FUNCTION_BLOCK FB_Teltonika

VAR_IN_OUT CONSTANT
	st_params	: st_Router_Params;
END_VAR

VAR_IN_OUT
	st_service : ST_router_service;
END_VAR

VAR
	realconverter : dwtoreal;
	w_SendSMS: WORD;
	set : st_router_set;
	ui_counter	:	uint;
END_VAR
VAR_OUTPUT
	Get	:	st_router_get;
END_VAR
VAR
	MBRead			: 	FB_MBReadRegs;
	MBWrite			:	FB_MBWriteRegs;
	MBSingleWrite	:	FB_MBWriteSingleReg;
	
	arw_DataBuffer		: 	ARRAY[0..62] OF word;
	st_WriteSMSData		:	STRING(20);

	ar_SMSData			:	ARRAY[0..89] OF WORD;
	ar_ReadSMSData		:	ARRAY[0..89] OF WORD;
	
	tempbuffer			:	ARRAY[0..10] OF WORD;

	
	ton_GetDataTimer				:	TON := (PT := TIME#1000MS);
	ton_StartSMSServiceDelay		:	TON := (PT := T#60S);

	
	ftrig_TransmissionDone	:	F_trig;
	
	ui_MBRetryCount			:	UINT;
	ui_SMSRetryCounter	:	UINT;
		
	ui_ForCounter	:	UINT;
	ui_MessageCounter	:	UINT;
	b_busy: BOOL;
	b_CommError: BOOL;
	udi_errid: UDINT;
	udi_cbread: UDINT;
	
	
	TempDTString	:	String;
END_VAR


VAR_IN_OUT
	s_Message	:	ARRAY[*] OF STRING;
END_VAR

VAR_INPUT
	s_SerialNumber		: STRING;
END_VAR

VAR CONSTANT
	e_ID 				: eObject_ID := eObject_ID.Router;
END_VAR

ton_GetDataTimer(IN:=NOT ton_GetDataTimer.Q);
ton_StartSMSServiceDelay();

ReadDataSFC();

get.Events.b_MBCommWarning := ui_MBRetryCount > 20;


//temporary setup via stparams until hmi setup is implemented.
set := st_params.ManualSettings;

ACTION aCheckAlarmMessages:
IF ton_StartSMSServiceDelay.Q THEN
	IF get.e_SMSStatus = eSMSStatus.Idle OR get.e_SMSStatus = eSMSStatus.error THEN
		//skip through message array until non_empty value or the end of the list is found 
		WHILE (s_Message[ui_MessageCounter] = '') AND (ui_MessageCounter < UPPER_BOUND(s_message, 1)) DO
			ui_MessageCounter := ui_MessageCounter + 1;
		END_WHILE
		
		IF (s_Message[ui_MessageCounter] <> '') THEN
			CreateMessage(s_Message[ui_MessageCounter]);	//check for valid message
			get.e_SMSStatus := eSMSStatus.NewMessage;
			s_Message[ui_MessageCounter] := '';
		END_IF
		
		IF ui_MessageCounter >= UPPER_BOUND(s_message, 1) THEN
			ui_MessageCounter := DINT_TO_UINT(LOWER_BOUND(s_message, 1)); 
		END_IF
	END_IF
END_IF
END_ACTION

ACTION aNetworkinfo:
MBRead(
	sIPAddr := st_params.IP_TELTONIKA,
	nTCPPort := st_params.MBPort_TELTONIKA,
	nUnitID := 1,
	nMBAddr := 103,
	nQuantity := 32,//*2,
	cbLength := SIZEOF(arw_DataBuffer),
	pDestAddr := ADR(arw_DataBuffer),
	bExecute := ton_GetDataTimer.Q,
	bBusy => b_busy,
	bError => b_CommError,
	nErrId => udi_errid,
	cbRead => udi_cbread,
	tTimeout := st_params.T_MBTimeout
);

ftrig_TransmissionDone(clk := b_busy);

IF ftrig_TransmissionDone.q THEN
	IF NOT b_CommError THEN
		FOR ui_ForCounter := 0 TO 31 DO
			arw_DataBuffer[ui_ForCounter] := be16_TO_HOST(arw_DataBuffer[ui_ForCounter]);
		END_FOR
		
		MEMCPY(ADR(Get.Mobile.NetworkInfo),  ADR(arw_DataBuffer[0]), 32);
		MEMCPY(ADR(Get.Mobile.NetworkType),  ADR(arw_DataBuffer[16]), 32);
		ui_MBRetryCount := 0;
		sfctip := TRUE;
	ELSE
		ui_MBRetryCount := ui_MBRetryCount + 1;
		sfctip := TRUE;
	END_IF
END_IF
END_ACTION

ACTION aReadActiveSim:

MBRead(
	sIPAddr := st_params.IP_TELTONIKA,
	nTCPPort := st_params.MBPort_TELTONIKA,
	nUnitID := 1,
	nMBAddr := 205,
	nQuantity := 1,//*2,
	cbLength := SIZEOF(arw_DataBuffer),
	pDestAddr := ADR(arw_DataBuffer),
	bExecute := ton_GetDataTimer.Q,
	bBusy => b_busy,
	bError => b_CommError,
	nErrId => udi_errid,
	cbRead => udi_cbread,
	tTimeout := st_params.T_MBTimeout
);

ftrig_TransmissionDone(clk := b_busy);

IF ftrig_TransmissionDone.q THEN
	IF NOT b_CommError THEN
	
		//Get.Mobile.ui_ActiveSim := arw_DataBuffer[0];
	
		ui_MBRetryCount := 0;
		sfctip := TRUE;
	ELSE
		ui_MBRetryCount := ui_MBRetryCount + 1;
		sfctip := TRUE;
	END_IF
END_IF
END_ACTION

ACTION aReadDataUsageSim1:

MBRead(
	sIPAddr := st_params.IP_TELTONIKA,
	nTCPPort := st_params.MBPort_TELTONIKA,
	nUnitID := 1,
	nMBAddr := 193,
	nQuantity := 4,//*2,
	cbLength := SIZEOF(arw_DataBuffer),
	pDestAddr := ADR(arw_DataBuffer),
	bExecute := ton_GetDataTimer.Q,
	bBusy => b_busy,
	bError => b_CommError,
	nErrId => udi_errid,
	cbRead => udi_cbread,
	tTimeout := st_params.T_MBTimeout
);

ftrig_TransmissionDone(clk := b_busy);

IF ftrig_TransmissionDone.q THEN
	IF NOT b_CommError THEN
	
		MEMCPY(ADR(Get.Mobile.ui_Sim1DataReceivedMonth)+2, ADR(arw_DataBuffer[0]), 2);
		MEMCPY(ADR(Get.Mobile.ui_Sim1DataReceivedMonth), ADR(arw_DataBuffer[1]), 2);
		
		MEMCPY(ADR(Get.Mobile.ui_Sim1DataSendMonth)+2, ADR(arw_DataBuffer[2]), 2);
		MEMCPY(ADR(Get.Mobile.ui_Sim1DataSendMonth), ADR(arw_DataBuffer[3]), 2);	
	
		ui_MBRetryCount := 0;
		sfctip := TRUE;
	ELSE
		ui_MBRetryCount := ui_MBRetryCount + 1;
		sfctip := TRUE;
	END_IF
END_IF
END_ACTION

ACTION aReadDataUsageSim2:

MBRead(
	sIPAddr := st_params.IP_TELTONIKA,
	nTCPPort := st_params.MBPort_TELTONIKA,
	nUnitID := 1,
	nMBAddr := 308,
	nQuantity := 4,//*2,
	cbLength := SIZEOF(arw_DataBuffer),
	pDestAddr := ADR(arw_DataBuffer),
	bExecute := ton_GetDataTimer.Q,
	bBusy => b_busy,
	bError => b_CommError,
	nErrId => udi_errid,
	cbRead => udi_cbread,
	tTimeout := st_params.T_MBTimeout
);

ftrig_TransmissionDone(clk := b_busy);

IF ftrig_TransmissionDone.q THEN
	IF NOT b_CommError THEN
	
		MEMCPY(ADR(Get.Mobile.ui_Sim2DataReceivedMonth)+2, ADR(arw_DataBuffer[0]), 2);
		MEMCPY(ADR(Get.Mobile.ui_Sim2DataReceivedMonth), ADR(arw_DataBuffer[1]), 2);
		
		MEMCPY(ADR(Get.Mobile.ui_Sim2DataSendMonth)+2, ADR(arw_DataBuffer[2]), 2);
		MEMCPY(ADR(Get.Mobile.ui_Sim2DataSendMonth), ADR(arw_DataBuffer[3]), 2);	
	
		ui_MBRetryCount := 0;
		sfctip := TRUE;
	ELSE
		ui_MBRetryCount := ui_MBRetryCount + 1;
		sfctip := TRUE;
	END_IF
END_IF
END_ACTION

ACTION AReadGeneral:

MBRead(
	sIPAddr := st_params.IP_TELTONIKA,
	nTCPPort := st_params.MBPort_TELTONIKA,
	nUnitID := 1,
	nMBAddr := 1,
	nQuantity := 6,//*2,
	cbLength := SIZEOF(arw_DataBuffer),
	pDestAddr := ADR(arw_DataBuffer),
	bExecute := ton_GetDataTimer.Q,
	bBusy => b_busy,
	bError => b_CommError,
	nErrId => udi_errid,
	cbRead => udi_cbread,
	tTimeout := st_params.T_MBTimeout
);

ftrig_TransmissionDone(clk := b_busy);

IF ftrig_TransmissionDone.q THEN
	IF NOT b_CommError THEN
		
		get.Device.SystemUptime :=	SHL(	WORD_TO_UDINT(	arw_DataBuffer[0]),16)	+	arw_DataBuffer[1];
		MEMCPY(ADR(Get.Mobile.RSSI)+2,  ADR(arw_DataBuffer[2]), 2);
		MEMCPY(ADR(Get.Mobile.RSSI),  ADR(arw_DataBuffer[3]), 2);

		//MEMCPY(ADR(Get.Mobile.NetworkOperator),  ADR(arw_DataBuffer[22]), 32);
		
		get.Device.Temperature	:= 	UDINT_TO_REAL ( SHL(	WORD_TO_UDINT(	arw_DataBuffer[4]),16)	+	arw_DataBuffer[5] )/10;

		ui_MBRetryCount := 0;
		sfctip := TRUE;
	ELSE
		ui_MBRetryCount := ui_MBRetryCount + 1;
		sfctip := TRUE;
	END_IF
END_IF
END_ACTION

ACTION aReadGPSData:


MBRead(
	sIPAddr := st_params.IP_TELTONIKA,
	nTCPPort := st_params.MBPort_TELTONIKA,
	nUnitID := 1,
	nMBAddr := 143,
	nQuantity := 42,//*2,
	cbLength := SIZEOF(arw_DataBuffer),
	pDestAddr := ADR(arw_DataBuffer),
	bExecute := ton_GetDataTimer.Q,
	bBusy => b_busy,
	bError => b_CommError,
	nErrId => udi_errid,
	cbRead => udi_cbread,
	tTimeout := st_params.T_MBTimeout
);

ftrig_TransmissionDone(clk := b_busy);

IF ftrig_TransmissionDone.q THEN
	IF NOT b_CommError THEN
		
		realconverter.Registers[2] := arw_DataBuffer[0];
		realconverter.Registers[1] := arw_DataBuffer[1];
		Get.GPS.Latitude  := realconverter.realvalue;
 
		realconverter.Registers[2] := arw_DataBuffer[2];
		realconverter.Registers[1] := arw_DataBuffer[3];
		Get.GPS.Longitude  := realconverter.realvalue;
		
		FOR ui_ForCounter := 4 TO 35 DO
			arw_DataBuffer[ui_ForCounter] := be16_TO_HOST(arw_DataBuffer[ui_ForCounter]);
		END_FOR
				
		MEMCPY(ADR(Get.GPS.FixTime),  ADR(arw_DataBuffer[4]), 32);			//GPS fixtime (text, unix timetamp * 1000)
						
		MEMCPY(ADR(TempDTString), ADR(arw_DataBuffer[20]), 32);			//GPS DateTime (text, YYYY-MM-DD HH:MM:SS)
		FindAndReplaceChar(ADR(TempDTString), ' ', '-', ADR(TempDTString), SIZEOF(TempDTString));	//replace space between date and time with dash
		TempDTString := concat(TempDTString, '.000');	//add milliseconds to string
		get.GPS.DateTime := SystemTime_TO_DT(String_TO_Systemtime(TempDTString));
		
		realconverter.Registers[2] := arw_DataBuffer[36];					//GPS speed
		realconverter.Registers[1] := arw_DataBuffer[37];
		Get.GPS.Speed  := realconverter.realvalue;
		
	
		MEMCPY(ADR(Get.GPS.SatCount)+2, ADR(arw_DataBuffer[38]), 2);			//GPS sattelite count
		MEMCPY(ADR(Get.GPS.SatCount), ADR(arw_DataBuffer[39]), 2);			//GPS sattelite count
		
		realconverter.Registers[2] := arw_DataBuffer[40];
		realconverter.Registers[1] := arw_DataBuffer[41];
		Get.GPS.Accuracy  := realconverter.realvalue;						//GPS accuracy
		
			
		ui_MBRetryCount := 0;
		sfctip := TRUE;
	ELSE
		ui_MBRetryCount := ui_MBRetryCount + 1;
		sfctip := TRUE;
	END_IF
END_IF
END_ACTION

ACTION aReadSerial:
MBRead(
	sIPAddr := st_params.IP_TELTONIKA,
	nTCPPort := st_params.MBPort_TELTONIKA,
	nUnitID := 1,
	nMBAddr := 39,
	nQuantity := 16,//*2,
	cbLength := SIZEOF(arw_DataBuffer),
	pDestAddr := ADR(arw_DataBuffer),
	bExecute := ton_GetDataTimer.Q,
	bBusy => b_busy,
	bError => b_CommError,
	nErrId => udi_errid,
	cbRead => udi_cbread,
	tTimeout := st_params.T_MBTimeout
);

ftrig_TransmissionDone(clk := b_busy);

IF ftrig_TransmissionDone.q THEN
	IF NOT b_CommError THEN
		FOR ui_ForCounter := 0 TO 16 DO
			arw_DataBuffer[ui_ForCounter] := be16_TO_HOST(arw_DataBuffer[ui_ForCounter]);
		END_FOR
		
		//MEMCPY(ADR(Get.Mobile.NetworkOperator),  ADR(arw_DataBuffer[0]), 32);
		MEMCPY(ADR(Get.Device.RouterSerial),  ADR(arw_DataBuffer[0]), 32);
		
		ui_MBRetryCount := 0;
		sfctip := TRUE;
	ELSE
		ui_MBRetryCount := ui_MBRetryCount + 1;
		sfctip := TRUE;
	END_IF
END_IF
END_ACTION

ACTION aSendSMS:

IF get.e_SMSStatus = eSMSStatus.SendingMessage THEN
	MBSingleWrite(
		sIPAddr := st_params.IP_TELTONIKA,
		nTCPPort := st_params.MBPort_TELTONIKA,
		nUnitID := 1,
		nMBAddr := 396,
		nValue	:=	1,
		bExecute := ton_GetDataTimer.Q,
		bBusy => b_busy,
		bError => b_CommError,
		nErrId => udi_errid,
		tTimeout := st_params.T_MBTimeout
	);
	
	ftrig_TransmissionDone(clk := b_busy);
	
	IF ftrig_TransmissionDone.q THEN
		IF NOT b_CommError THEN
			get.e_SMSStatus := eSMSSTatus.idle;		
			ui_SMSRetryCounter := 0;
			ui_MBRetryCount := 0;
			sfctip := TRUE;
		ELSE
			ui_MBRetryCount := ui_MBRetryCount + 1;
			ui_SMSRetryCounter := ui_SMSRetryCounter + 1;
			IF ui_SMSRetryCounter > 0 THEN
				get.Events.b_SMSNotSendError := TRUE;
				get.e_SMSStatus := eSMSStatus.error;
				sfctip := TRUE;
			END_IF
		END_IF
	END_IF
ELSE
	SFCtip := NOT SFCTip;
END_IF
END_ACTION

ACTION aWriteSimSettings:

arw_DataBuffer[0] := TO_UINT(set.SimSelectionMode);
arw_DataBuffer[1] := TO_UINT(set.Sim1Pin);
arw_DataBuffer[2] := TO_UINT(set.Sim2Pin);

//FOR ui_counter := 1 TO 3 DO
//	arw_DataBuffer[ui_counter] := host_to_be16(arw_DataBuffer[ui_counter]);
//END_FOR

MBWrite(
	sIPAddr := st_params.IP_TELTONIKA,
	nTCPPort := st_params.MBPort_TELTONIKA,
	nUnitID := 1,
	nMBAddr := 1049,
	nQuantity := 3,
	cbLength := SIZEOF(arw_DataBuffer),
	pSrcAddr	:=	ADR(arw_DataBuffer),
	bExecute := ton_GetDataTimer.Q,
	bBusy => b_busy,
	bError => b_CommError,
	nErrId => udi_errid,
	tTimeout := st_params.T_MBTimeout
);

ftrig_TransmissionDone(clk := b_busy);

IF ftrig_TransmissionDone.q THEN
		sfctip := TRUE;
END_IF
END_ACTION

ACTION aWriteSMSData:

MBWrite(
	sIPAddr := st_params.IP_TELTONIKA,
	nTCPPort := st_params.MBPort_TELTONIKA,
	nUnitID := 1,
	nMBAddr := 397,
	nQuantity := 90,
	cbLength := SIZEOF(ar_SMSData),
	pSrcAddr	:=	ADR(ar_SMSData),
	bExecute := ton_GetDataTimer.Q,
	bBusy => b_busy,
	bError => b_CommError,
	nErrId => udi_errid,
	tTimeout := st_params.T_MBTimeout
);

ftrig_TransmissionDone(clk := b_busy);

IF ftrig_TransmissionDone.q THEN
	IF NOT b_CommError THEN
		get.e_SMSStatus := eSMSStatus.SendingMessage;
		ui_SMSRetryCounter := 0;
		ui_MBRetryCount := 0;
		sfctip := TRUE;
	ELSE
		ui_SMSRetryCounter := ui_SMSRetryCounter +1;
		ui_MBRetryCount := ui_MBRetryCount + 1;
		IF ui_SMSRetryCounter > 3 THEN
			get.Events.b_SMSNotSendError := TRUE;
			get.e_SMSStatus := eSMSStatus.error;
			sfctip := TRUE;
		END_IF
	END_IF
END_IF
END_ACTION

ACTION Bypass_active:
get.e_SMSStatus := eSMSStatus.Idle;
get.Events.b_SMSNotSendError := FALSE;
END_ACTION

METHOD CreateMessage : BOOL
VAR_INPUT
//	TelNumber	:	ULINT;
	s_Message		:	STRING(80);
END_VAR

VAR
	s_InternalMessage 	: 	STRING(160);
	s_LAT				:	STRING(8);
	s_LONG				:	STRING(9);
	ui_counter			:	UINT;
END_VAR
IF NOT get.Events.b_NoSMSNumberAvailable THEN
	memcpy(ADR(ar_SMSData[0]), ADR(get.Mobile.s_EmergencySMSNumber), 20);
	
	s_LAT := REAL_TO_STRING(get.GPS.Latitude);
	s_LONG := REAL_TO_STRING(get.GPS.Longitude);
	
	s_InternalMessage := 'ePU10 LFP Battery System';
	s_InternalMessage := concat(s_InternalMessage, '$n');
	s_InternalMessage := concat(s_InternalMessage, 'ID: ');
	s_InternalMessage := concat(s_InternalMessage, get.mobile.s_EmergencySMSDevName);
	s_InternalMessage := concat(s_InternalMessage, '$n');
	s_InternalMessage := concat(s_InternalMessage, 'LAT: ');
	s_InternalMessage := concat(s_InternalMessage, s_LAT);
	s_InternalMessage := concat(s_InternalMessage, '$n');
	s_InternalMessage := concat(s_InternalMessage, 'LON: ');
	s_InternalMessage := concat(s_InternalMessage, s_LONG);
	s_InternalMessage := concat(s_InternalMessage, '$n');
	s_InternalMessage := concat(s_InternalMessage,s_Message);
	
	memcpy(ADR(ar_SMSData[10]), ADR(s_InternalMessage[0]), 160);
	
	FOR ui_counter := 0 TO 89 DO
		ar_SMSData[ui_counter] := host_to_be16(ar_SMSData[ui_counter]);
	END_FOR

	CreateMessage := TRUE;
ELSE
	get.Events.b_SMSNotSendError := TRUE;
	CreateMessage := TRUE;
END_IF
END_METHOD

METHOD EMStop : BOOL
VAR_INPUT
END_VAR

//nothing to do here
EMSTOP := TRUE;
END_METHOD

METHOD FB_init : BOOL
VAR_INPUT
	bInitRetains : BOOL; // if TRUE, the retain variables are initialized (warm start / cold start)
	bInCopyCode : BOOL;  // if TRUE, the instance afterwards gets moved into the copy code (online change)
END_VAR
ton_StartSMSServiceDelay(IN := TRUE);
END_METHOD

METHOD GetDiagnostics : BOOL
VAR_IN_OUT
	AddError		: ARRAY [*] OF FB_AddErrorST;
	a_ActiveEvents	: ARRAY [*] OF ST_ErrorStruct;
	w_Index			: WORD;
END_VAR
(*No emergency number configured*)	AddError[w_Index](
			b_ErrorTrig				:= get.Events.b_NoSMSNumberAvailable,
			b_SMSEnableVDL			:= FALSE,
			out_ST_Error			:= a_ActiveEvents[w_Index],
			w_ErrorID				:= 1,
			e_ObjectID				:= e_id,						//only first call set object ID.
			s_Message				:= 'no sms number available',
			e_sev					:= eSeverity.info,
			b_AutoClear				:= TRUE,
			e_ErrAckAccess			:= eErrAckAccess.General
			);
		w_Index := w_Index +1;
		
(*SMS not send warning*)	AddError[w_Index](
			b_ErrorTrig				:= get.Events.b_SMSNotSendError,
			b_SMSEnableVDL			:= FALSE,
			out_ST_Error			:= a_ActiveEvents[w_Index],
			w_ErrorID				:= 2,					
			s_Message				:= 'SMS not send',
			e_sev					:= eSeverity.info,
			b_AutoClear				:= TRUE,
			t_triggerTime			:= T#10S,
			e_ErrAckAccess			:= eErrAckAccess.General
			);
		w_Index := w_Index +1;
		
(*Modbus comm warning*)	AddError[w_Index](
			b_ErrorTrig				:= get.Events.b_MBCommWarning,
			b_SMSEnableVDL			:= FALSE,
			out_ST_Error			:= a_ActiveEvents[w_Index],
			w_ErrorID				:= 3,					
			s_Message				:= 'modbus comm. warning',
			e_sev					:= eSeverity.warning,
			b_AutoClear				:= TRUE,
			e_ErrAckAccess			:= eErrAckAccess.General
			);
		w_Index := w_Index +1;
		
(*GPS location missing*)	AddError[w_Index](
			b_ErrorTrig				:= get.Events.b_noGPSFixWarning,
			b_SMSEnableVDL			:= FALSE,
			out_ST_Error			:= a_ActiveEvents[w_Index],
			w_ErrorID				:= 5,					
			s_Message				:= 'no gps location available',
			e_sev					:= eSeverity.info,
			b_AutoClear				:= TRUE,
			e_ErrAckAccess			:= eErrAckAccess.General
			);
		w_Index := w_Index +1;
		
(*network missing*)	AddError[w_Index](
			b_ErrorTrig				:= get.Events.b_NoNetworkWarning,
			b_SMSEnableVDL			:= FALSE,
			out_ST_Error			:= a_ActiveEvents[w_Index],
			w_ErrorID				:= 6,					
			s_Message				:= 'no network available',
			e_sev					:= eSeverity.info,
			b_AutoClear				:= TRUE,
			e_ErrAckAccess			:= eErrAckAccess.General
			);
		w_Index := w_Index +1;
		
(*simcard missing*)	AddError[w_Index](
			b_ErrorTrig				:= get.Events.b_NoSimWarning,
			b_SMSEnableVDL			:= FALSE,
			out_ST_Error			:= a_ActiveEvents[w_Index],
			w_ErrorID				:= 7,					
			s_Message				:= 'no simcard available',
			e_sev					:= eSeverity.info,
			b_AutoClear				:= TRUE,
			e_ErrAckAccess			:= eErrAckAccess.General
			);
		w_Index := w_Index +1;
END_METHOD

ACTION ReadCustomRegisters:

MBRead(
	sIPAddr := st_params.IP_TELTONIKA,
	nTCPPort := st_params.MBPort_TELTONIKA,
	nUnitID := 1,
	nMBAddr := 1024,
	nQuantity := 7,//*2,
	cbLength := SIZEOF(arw_DataBuffer),
	pDestAddr := ADR(arw_DataBuffer),
	bExecute := ton_GetDataTimer.Q,
	bBusy => b_busy,
	bError => b_CommError,
	nErrId => udi_errid,
	cbRead => udi_cbread,
	tTimeout := st_params.T_MBTimeout
);

ftrig_TransmissionDone(clk := b_busy);

IF ftrig_TransmissionDone.q THEN
	IF NOT b_CommError THEN
		get.Mobile.ui_ActiveSim 		:= 	arw_DataBuffer[0];
		get.Mobile.SimStatus 			:= 	arw_DataBuffer[1];
		get.Mobile.ModemState 			:= 	arw_DataBuffer[2];
		get.Mobile.NetworkState 		:=  arw_DataBuffer[3];
		get.Wifi.WifiClienModeStatus 	:= 	arw_DataBuffer[4]; 
		get.Wifi.WifiAPModeStatus 		:= 	arw_DataBuffer[5]; 		//not yet implemented
		get.Wifi.WifiApNumberOfClients 	:= 	arw_DataBuffer[6]; 
		
			
		ui_MBRetryCount := 0;
		sfctip := TRUE;
	ELSE
		ui_MBRetryCount := ui_MBRetryCount + 1;
		sfctip := TRUE;
	END_IF
END_IF
END_ACTION

ACTION ReadDataSFC:
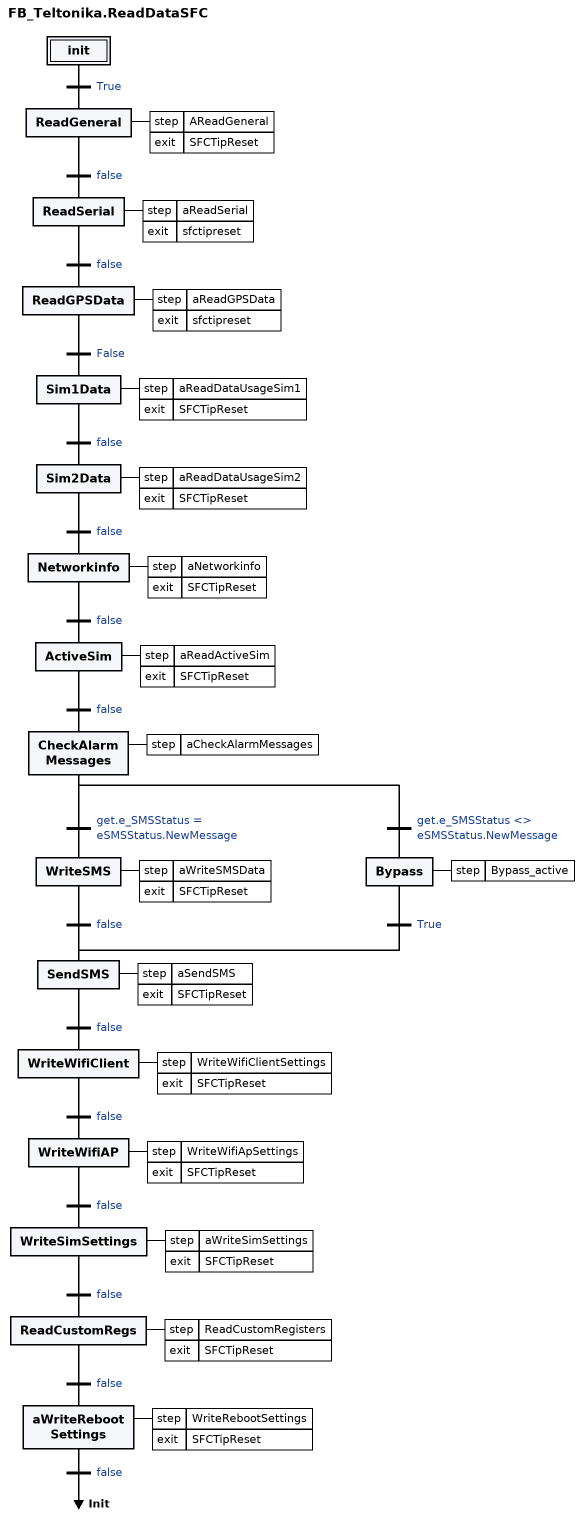
INITIAL_STEP init:
END_STEP
TRANSITION FROM init TO ReadGeneral
    := True;
END_TRANSITION
STEP ReadGeneral:
    AReadGeneral(N);  // step action
    SFCTipReset(P0);  // exit action
END_STEP
TRANSITION FROM ReadGeneral TO ReadSerial
    := false;
END_TRANSITION
STEP ReadSerial:
    aReadSerial(N);  // step action
    sfctipreset(P0);  // exit action
END_STEP
TRANSITION FROM ReadSerial TO ReadGPSData
    := false;
END_TRANSITION
STEP ReadGPSData:
    aReadGPSData(N);  // step action
    sfctipreset(P0);  // exit action
END_STEP
TRANSITION FROM ReadGPSData TO Sim1Data
    := False;
END_TRANSITION
STEP Sim1Data:
    aReadDataUsageSim1(N);  // step action
    SFCTipReset(P0);  // exit action
END_STEP
TRANSITION FROM Sim1Data TO Sim2Data
    := false;
END_TRANSITION
STEP Sim2Data:
    aReadDataUsageSim2(N);  // step action
    SFCTipReset(P0);  // exit action
END_STEP
TRANSITION FROM Sim2Data TO Networkinfo
    := false;
END_TRANSITION
STEP Networkinfo:
    aNetworkinfo(N);  // step action
    SFCTipReset(P0);  // exit action
END_STEP
TRANSITION FROM Networkinfo TO ActiveSim
    := false;
END_TRANSITION
STEP ActiveSim:
    aReadActiveSim(N);  // step action
    SFCTipReset(P0);  // exit action
END_STEP
TRANSITION FROM ActiveSim TO CheckAlarmMessages
    := false;
END_TRANSITION
STEP CheckAlarmMessages:
    aCheckAlarmMessages(N);  // step action
END_STEP
TRANSITION FROM CheckAlarmMessages TO WriteSMS
    := get.e_SMSStatus = eSMSStatus.NewMessage;
END_TRANSITION
STEP WriteSMS:
    aWriteSMSData(N);  // step action
    SFCTipReset(P0);  // exit action
END_STEP
TRANSITION FROM WriteSMS TO SendSMS
    := false;
END_TRANSITION
TRANSITION FROM CheckAlarmMessages TO Bypass
    := get.e_SMSStatus <> eSMSStatus.NewMessage;
END_TRANSITION
STEP Bypass:
    Bypass_active(N);  // step action
END_STEP
TRANSITION FROM Bypass TO SendSMS
    := True;
END_TRANSITION
STEP SendSMS:
    aSendSMS(N);  // step action
    SFCTipReset(P0);  // exit action
END_STEP
TRANSITION FROM SendSMS TO WriteWifiClient
    := false;
END_TRANSITION
STEP WriteWifiClient:
    WriteWifiClientSettings(N);  // step action
    SFCTipReset(P0);  // exit action
END_STEP
TRANSITION FROM WriteWifiClient TO WriteWifiAP
    := false;
END_TRANSITION
STEP WriteWifiAP:
    WriteWifiApSettings(N);  // step action
    SFCTipReset(P0);  // exit action
END_STEP
TRANSITION FROM WriteWifiAP TO WriteSimSettings
    := false;
END_TRANSITION
STEP WriteSimSettings:
    aWriteSimSettings(N);  // step action
    SFCTipReset(P0);  // exit action
END_STEP
TRANSITION FROM WriteSimSettings TO ReadCustomRegs
    := false;
END_TRANSITION
STEP ReadCustomRegs:
    ReadCustomRegisters(N);  // step action
    SFCTipReset(P0);  // exit action
END_STEP
TRANSITION FROM ReadCustomRegs TO aWriteRebootSettings
    := false;
END_TRANSITION
STEP aWriteRebootSettings:
    WriteRebootSettings(N);  // step action
    SFCTipReset(P0);  // exit action
END_STEP
TRANSITION FROM aWriteRebootSettings TO Init
    := false;
END_TRANSITION
// branch label Branch0_ReadDataSFC
END_ACTION

METHOD Reset : BOOL
VAR_INPUT
END_VAR
get.Events.b_SMSNotSendError := FALSE;
get.e_SMSStatus := eSMSStatus.Idle;

Reset := TRUE;
END_METHOD

METHOD SetDevName : BOOL
VAR_INPUT
	s_DevName	:	String(12);
END_VAR
IF s_DevName = '' THEN
	get.Mobile.s_EmergencySMSDevName := ''; //<-- stParams.serial number
ELSE
	get.Mobile.s_EmergencySMSDevName :=	s_DevName;
END_IF

SetDevName := get.Mobile.s_EmergencySMSDevName <> '';
END_METHOD

METHOD SetSMSNumber : BOOL
VAR_INPUT
	s_SMSNumber	:	STRING(20);
END_VAR
VAR 
	for_counter	:	UINT :=0;
	InternalString	:	STRING(20);
	intermediateValue	:	UINT;
	
	temp	:	string(10);
END_VAR

SetSMSNumber := TRUE;

//check minimum length
IF INT_TO_UINT(len(s_SMSNumber)) < st_params.MinimumPhoneNumberLength AND s_SMSNumber <> '' THEN
	SetSMSNumber := FALSE;
ELSE
	InternalString := s_SMSNumber;
	
	//replace leading + with 00
	IF left(InternalString,1) = '+' THEN
		InternalString := Replace(InternalString, '00', 1, 1);
	END_IF
	
	//check for non_numeric characters
	FOR for_counter := 1 TO INT_TO_UINT(len(InternalString)) DO
		intermediateValue := f_toASC(mid(InternalString, 1, UINT_TO_INT(for_counter)));
		IF (intermediateValue < 48 OR intermediateValue > 57) THEN
			SetSMSNumber := FALSE;
		END_IF
	END_FOR
END_IF

//only if all checks succeed, the number is written to the struct.
IF SetSMSNumber THEN
	get.Mobile.s_EmergencySMSNumber := InternalString;
ELSE
	get.Mobile.s_EmergencySMSNumber := '';
END_IF

get.Events.b_NoSMSNumberAvailable := NOT SetSMSNumber;
END_METHOD

ACTION SFCTipReset:
SFCTip := FALSE;
END_ACTION

ACTION WriteRebootSettings:

arw_DataBuffer[0] := TO_UINT(set.AutoRebootEnable);
arw_DataBuffer[1] := TO_UINT(set.ManualReboot);

MBWrite(
	sIPAddr := st_params.IP_TELTONIKA,
	nTCPPort := st_params.MBPort_TELTONIKA,
	nUnitID := 1,
	nMBAddr := 1139,
	nQuantity := 2,
	cbLength := SIZEOF(arw_DataBuffer),
	pSrcAddr	:=	ADR(arw_DataBuffer),
	bExecute := ton_GetDataTimer.Q,
	bBusy => b_busy,
	bError => b_CommError,
	nErrId => udi_errid,
	tTimeout := st_params.T_MBTimeout
);

ftrig_TransmissionDone(clk := b_busy);

IF ftrig_TransmissionDone.q THEN
	sfctip := TRUE;
	set.ManualReboot := false;
END_IF
END_ACTION

ACTION WriteWifiAPSettings:

arw_DataBuffer[0] := TO_UINT(set.EnableWifiAP);
memcpy(ADR(arw_DataBuffer[1]), ADR(set.WifiAPSSID), 32);
memcpy(ADR(arw_DataBuffer[17]), ADR(set.WifiAPPass), 32);
arw_DataBuffer[33] := TO_UINT(set.WifiAPSecType);

FOR ui_counter := 1 TO 32 DO
	arw_DataBuffer[ui_counter] := host_to_be16(arw_DataBuffer[ui_counter]);
END_FOR

MBWrite(
	sIPAddr := st_params.IP_TELTONIKA,
	nTCPPort := st_params.MBPort_TELTONIKA,
	nUnitID := 1,
	nMBAddr := 1099,
	nQuantity := 34,
	cbLength := SIZEOF(arw_DataBuffer),
	pSrcAddr	:=	ADR(arw_DataBuffer),
	bExecute := ton_GetDataTimer.Q,
	bBusy => b_busy,
	bError => b_CommError,
	nErrId => udi_errid,
	tTimeout := st_params.T_MBTimeout
);

ftrig_TransmissionDone(clk := b_busy);

IF ftrig_TransmissionDone.q THEN
		sfctip := TRUE;
END_IF
END_ACTION

ACTION WriteWifiClientSettings:

arw_DataBuffer[0] := TO_UINT(set.EnableWifiClient);
memcpy(ADR(arw_DataBuffer[1]), ADR(set.WifiClientSSID), 32);
memcpy(ADR(arw_DataBuffer[17]), ADR(set.WifiClientPass), 32);
arw_DataBuffer[33] := TO_UINT(set.WifiClientSecType);

FOR ui_counter := 1 TO 32 DO
	arw_DataBuffer[ui_counter] := host_to_be16(arw_DataBuffer[ui_counter]);
END_FOR

MBWrite(
	sIPAddr := st_params.IP_TELTONIKA,
	nTCPPort := st_params.MBPort_TELTONIKA,
	nUnitID := 1,
	nMBAddr := 1059,
	nQuantity := 34,
	cbLength := SIZEOF(arw_DataBuffer),
	pSrcAddr	:=	ADR(arw_DataBuffer),
	bExecute := ton_GetDataTimer.Q,
	bBusy => b_busy,
	bError => b_CommError,
	nErrId => udi_errid,
	tTimeout := st_params.T_MBTimeout
);

ftrig_TransmissionDone(clk := b_busy);

IF ftrig_TransmissionDone.q THEN
		sfctip := TRUE;
END_IF
END_ACTION

END_FUNCTION_BLOCK

(* stored: Version 1.1.0.1, ProductVersion 3.1.4026.18
   POU FB_Teltonika: Id {ce5c4c16-d731-4cac-8a46-0d3c64bd48ea}, SpecialFunc None
   Folder SFC: Id {f4d5eef4-c143-4170-8575-a31d9721c5b0}
   Action aCheckAlarmMessages: Id {8bb623ce-e32a-4247-9eea-59e963096791}
   Action aNetworkinfo: Id {d8e545ad-0207-4319-80fa-b51b970a255b}
   Action aReadActiveSim: Id {44a57084-24be-4d2d-b636-a258a594fbe8}
   Action aReadDataUsageSim1: Id {c47efe6a-5222-482b-8137-7d1c7960cdfe}
   Action aReadDataUsageSim2: Id {a46a9137-6bea-46c4-9399-6f8cdaede783}
   Action AReadGeneral: Id {fc40b227-86e2-44d0-8f40-6ded2a1905ff}
   Action aReadGPSData: Id {6c2c6e09-da82-480e-b334-1a203187c02b}
   Action aReadSerial: Id {709e3d7b-e520-4ed8-84a9-db04b277e3ea}
   Action aSendSMS: Id {6390c9e1-ff00-4b14-bfc1-4efb550b3995}
   Action aWriteSimSettings: Id {9027dbe8-5f04-4050-ab52-3b0e533410d9}
   Action aWriteSMSData: Id {f2cd87f2-3ec6-4b9a-960d-7ee9b04df6de}
   Action Bypass_active: Id {c9bfb550-60be-4a3e-953b-76d365f8ac6b}
   Method CreateMessage: Id {313919e7-6b12-4358-9d52-916d3392c894}
   Method EMStop: Id {6ba89e65-66e3-4e9c-adf4-3239c5d5f77d}
   Method FB_init: Id {1a01fa31-54b0-4def-ba42-8fd997b71ea0}
   Method GetDiagnostics: Id {40b6fdc8-4d98-479c-b936-17011da3130d}
   Action ReadCustomRegisters: Id {c7edffe8-6b37-4221-b04f-7a3c1515e057}
   Action ReadDataSFC: Id {4a4da098-fd72-47ce-861d-90616dad5bf0}
   Method Reset: Id {bd7c570d-38bf-480e-a9c9-2d2f0b0af6b7}
   Method SetDevName: Id {0b75bd53-ab4d-436d-b710-af600db034db}
   Method SetSMSNumber: Id {b87a798f-bceb-4992-bb50-ae879adcce42}
   Action SFCTipReset: Id {67752440-1bb6-4e7c-a33c-97f3b09a1c60}
   Action WriteRebootSettings: Id {ca462f55-809a-4b51-a0e3-f8e23f5e096d}
   Action WriteWifiAPSettings: Id {a7c28fe6-3bc4-439e-80ea-f2095b9a28ee}
   Action WriteWifiClientSettings: Id {86421294-3ba8-467c-9a1e-9f879966b621} *)
